Fanuc KAREL source: kd00035.KL

-- PROVISIONAL review KL for V770-1; original PC SHA256 4bc2b47c0d6212331c8fe27adad13785a4aa0d4e7a4724198289be6773343d5f
-- Incomplete behavior may be omitted. Consult companion uncertainty JSON. Do not deploy.
PROGRAM KD00035
%NOLOCKGROUP
VAR
  I : INTEGER
  J : INTEGER
  B : BOOLEAN
  R : REAL
  S : STRING[80]
BEGIN
  -- UNRESOLVED_PC offsets 5-18; opcodes 9D,81,18,9D,1B,9D,12,9C,13,04
  -- UNRESOLVED_PC offsets 23-27; opcodes 7F
END KD00035
